# EPICS StreamDevice protocol: code/10/geophone.proto
# ./wgsApp/Db/geophone.proto
Terminator = CR LF;
get_wf {
   ExtraInput = Ignore;
   replyTimeout=2000;
   out "WF?";
   separator=",";
   in "%f";
}
